TYPE ST_Shell :
STRUCT
	stPlatform		: ST_ShellPlatform;		(*  *)
	stFlags			: ST_ShellFlags;		(*  *)
	stRecipeData	: ST_ShellRecipeData;	(*  *)
END_STRUCT
END_TYPE

(* stored: Version 1.1.0.1, ProductVersion 3.1.4024.9
   DUT ST_Shell: Id {cf0d1b45-0bda-4ce4-9db2-5f6873174364} *)
